{attribute 'qualified_only'}
{attribute 'strict'}
TYPE cDeviceHeading :
// Various internal to station headings.
// Stations will use only appropriate headings for their station type
(
	
	Empty := 0,
	Puck := 1,
	Tray := 2,
	Carrier := 3,
	Tote := 4,
	Carton := 5,
	Box := 6,
	Buffer := 20,
	VisionStand := 10,
	ExceptionConv := 11,
	Flipper := 30,
	EvalToolType1 := 31,
	EvalToolType2 := 32,
	JustifyNest1 := 101,
	JustifyNest2 := 102,
	Reject := 998,
	Recovery := 999
	
) DINT;
END_TYPE

(* stored: Version 1.1.0.1, ProductVersion 3.1.4024.6
   DUT cDeviceHeading: Id {71b2a957-b05a-44aa-9955-60ed8bcda427} *)
